// Mitsubishi GX Works2 project: test   PLC: Q02U

PROGRAM MAIN
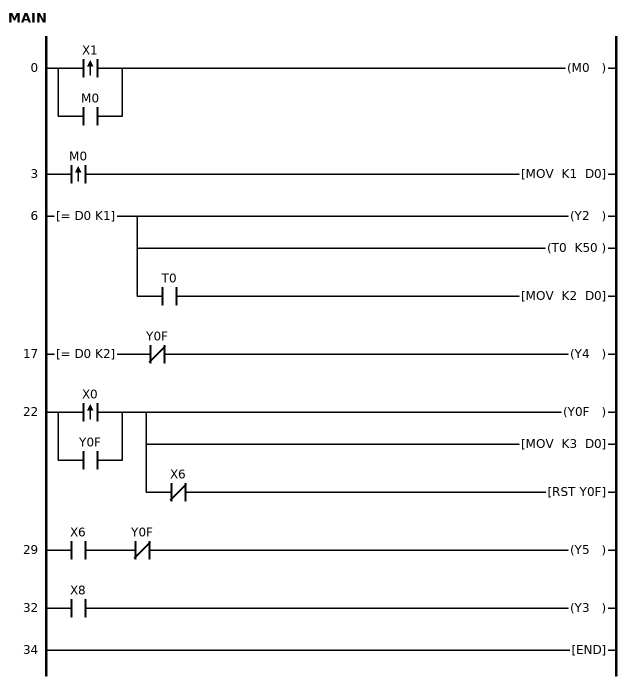
0     LDP     X1
      OR      M0
      OUT     M0
3     LDP     M0
      MOV     K1 D0
6     LD=     D0 K1
      OUT     Y2
      OUT     T0 K50
      AND     T0
      MOV     K2 D0
17    LD=     D0 K2
      ANI     Y0F
      OUT     Y4
22    LDP     X0
      OR      Y0F
      OUT     Y0F
      MOV     K3 D0
      ANI     X6
      RST     Y0F
29    LD      X6
      ANI     Y0F
      OUT     Y5
32    LD      X8
      OUT     Y3
34    END
END_PROGRAM
